// TIA Portal project "FactoryIO_Template_S7-1200_V15_V16" (V16)
// Vorlageprojekt für das Buch mit Zielsystem S7-1200

(* hardware
DEVICE "S7-1200-Station_1"  S7-1200 Station
   slot 0: "Baugruppenträger_0"  Rack  V1.0
   slot 1: "PLC_1"  CPU 1214C DC/DC/Rly  6ES7 214-1HG40-0XB0  V4.4
   slot 2: "DQ 16x24VDC_1"  SM 1222 DQ16 x 24VDC  6ES7 222-1BH32-0XB0  V2.0
*)

// ===== PLC "PLC_1"  CPU 1214C DC/DC/Rly =====

VAR_GLOBAL   // PLC tag table "Standard-Variablentabelle"
   "system" AT %M0.0 : Bool;
   "small_box_sensor_memory" AT %M0.1 : Bool;
   "large_box_sensor_memory" AT %M0.2 : Bool;
   "Transfer Right" AT %Q1.0 : Bool;
   "Tag_1" AT %M0.3 : Bool;
   "Tag_2" AT %M0.4 : Bool;
END_VAR

VAR_GLOBAL   // PLC tag table "Tag table from XML_1"
   "Start Button 1" AT %I0.0 : Bool;
   "Stop Button 1" AT %I0.1 : Bool;
   "Reset Button 1" AT %I0.2 : Bool;
   "Emergency Stop 1" AT %I0.3 : Bool;
   "input sensor" AT %I0.4 : Bool;
   "Roller Limit Sensor" AT %I0.5 : Bool;
   "Left Conveyor Sensor" AT %I0.6 : Bool;
   "Right Conveyor Sensor" AT %I0.7 : Bool;
   "Left Conveyor End Sensor" AT %I1.0 : Bool;
   "Right Conveyor End Sensor" AT %I1.1 : Bool;
   "Small Box Sensor" AT %I1.2 : Bool;
   "Large Box Sensor" AT %I1.3 : Bool;
   "Start Button Light" AT %Q0.0 : Bool;
   "Stop Button Light" AT %Q0.1 : Bool;
   "Reset Button Light" AT %Q0.2 : Bool;
   "Roller Conveyor (4m) 1" AT %Q0.3 : Bool;
   "Roller Conveyor (4m) 2" AT %Q0.4 : Bool;
   "Roller Conveyor (4m) 3" AT %Q0.5 : Bool;
   "roll forward" AT %Q0.6 : Bool;
   "Transfer Left" AT %Q0.7 : Bool;
   "Small Box Counter" AT %QD8 : DInt;
   "Large Box Counter" AT %QD12 : DInt;
END_VAR

// folder: System blocks/Program resources

DATA_BLOCK "IEC_Counter_0_DB"   // DB1
{ S7_Optimized_Access := 'TRUE' }
AUTHOR : Simatic
FAMILY : IEC
NAME : CNTR
VERSION : 1.0
// stored: InstanceOfName IEC_COUNTER
"IEC_COUNTER"
BEGIN
END_DATA_BLOCK

DATA_BLOCK "timer 2"   // DB2
{ S7_Optimized_Access := 'TRUE' }
AUTHOR : Simatic
FAMILY : IEC
NAME : IEC_TMR
VERSION : 1.0
// stored: InstanceOfName IEC_TIMER
"IEC_TIMER"
BEGIN
END_DATA_BLOCK

DATA_BLOCK "timer 1"   // DB3
{ S7_Optimized_Access := 'TRUE' }
AUTHOR : Simatic
FAMILY : IEC
NAME : IEC_TMR
VERSION : 1.0
// stored: InstanceOfName IEC_TIMER
"IEC_TIMER"
BEGIN
END_DATA_BLOCK

DATA_BLOCK "Counter 2"   // DB4
{ S7_Optimized_Access := 'TRUE' }
AUTHOR : Simatic
FAMILY : IEC
NAME : CNTR
VERSION : 1.0
// stored: InstanceOfName IEC_COUNTER
"IEC_COUNTER"
BEGIN
END_DATA_BLOCK

// folder: (top level)

FUNCTION "MHJ-PLC-Lab-Function-S71200" : Void   // FC9000, SCL
{ S7_Optimized_Access := 'TRUE' }
VERSION : 0.1
   VAR_TEMP
      rdTimeReturn : Int;
      outputTime : DTL;
      SyncVal : Byte;
      forVal : Int;
      forVal_2 : Int;
      Value : Byte;
   END_VAR
   VAR CONSTANT
      CompVal : Byte := 16#34;
      Value_01 : Byte := 16#11;
      Value_01_DW : DWord := 16#A165_D992;
      Value_02_DW : DWord := 16#58BE_4401;
   END_VAR
BEGIN

   #Value:=PEEK(area := 16#82,
        dbNumber := 0,
        byteOffset := 511);
   #Value := #Value + 1;

   POKE(area := 16#82,
        dbNumber := 0,
        byteOffset := 511,
        value := #Value);

   POKE(area:=16#81,
        dbNumber:=0,
        byteOffset:=1016,
        value:=#Value_01_DW);
   POKE(area := 16#81,
        dbNumber := 0,
        byteOffset := 1020,
        value := #Value_02_DW);

   POKE(area := 16#81,
        dbNumber := 0,
        byteOffset := 511,
        value := B#16#00);

   FOR #forVal := 0 TO 120 DO
       FOR #forVal_2:=0 TO 10 DO
           #rdTimeReturn:=RD_SYS_T(#outputTime);
           #rdTimeReturn := WR_SYS_T(#outputTime);
           #rdTimeReturn := RD_SYS_T(#outputTime);
           #rdTimeReturn := WR_SYS_T(#outputTime);
       END_FOR;
       #SyncVal:= PEEK(area := 16#81,
                      dbNumber := 0,
                      byteOffset := 511);
       IF #SyncVal = #CompVal THEN
          GOTO M_1;
       END_IF;
   END_FOR;
   RETURN;

   M_1:
   POKE(area := 16#81,
        dbNumber := 0,
        byteOffset := 511,
        value := B#16#0);
END_FUNCTION

ORGANIZATION_BLOCK "Main"   // OB1, LAD, ProgramCycle
TITLE = "Main Program Sweep (Cycle)"
{ S7_Optimized_Access := 'TRUE' }
VERSION : 0.1
   VAR_INPUT
      Initial_Call : Bool;   // Initial call of this OB
      Remanence : Bool;   // =True, if remanent data are available
   END_VAR
   VAR_TEMP   // added for the SCL form of the ladder/FBD networks
      _w1 : Bool;
   END_VAR
BEGIN

REGION Network 1: Konnektierungsbaustein für PLC-Lab
   // Im Netzwerk 1 wird der Konnektierungsbaustein für PLC-Lab aufgerufen.
   // Dieser Aufruf darf nicht entfernt werden!
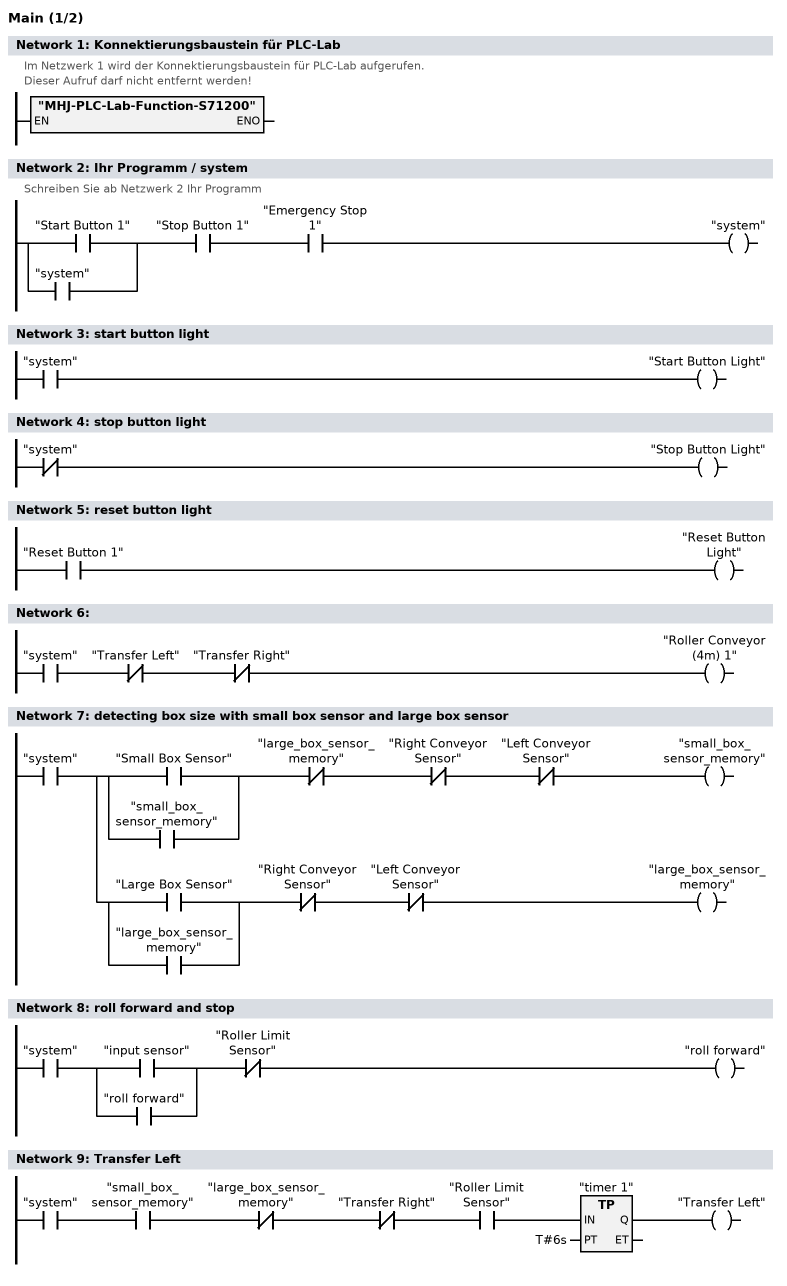
   RUNG wire#powerrail
      "MHJ-PLC-Lab-Function-S71200"()
   END_RUNG
   // the same network as SCL:
   "MHJ-PLC-Lab-Function-S71200"();
END_REGION

REGION Network 2: Ihr Programm / system
   // Schreiben Sie ab Netzwerk 2 Ihr Programm
   RUNG wire#powerrail
      Contact( "Start Button 1" )
      wire#w1
      Contact( "Stop Button 1" )
      Contact( "Emergency Stop 1" )
      Coil( "system" )
   END_RUNG
   RUNG wire#powerrail
      Contact( "system" )
   END_RUNG wire#w1
   // the same network as SCL:
   "system" := ("Start Button 1" OR "system") AND "Stop Button 1" AND "Emergency Stop 1";
END_REGION

REGION Network 3: start button light
   RUNG wire#powerrail
      Contact( "system" )
      Coil( "Start Button Light" )
   END_RUNG
   // the same network as SCL:
   "Start Button Light" := "system";
END_REGION

REGION Network 4: stop button light
   RUNG wire#powerrail
      I_Contact( "system" )
      Coil( "Stop Button Light" )
   END_RUNG
   // the same network as SCL:
   "Stop Button Light" := NOT "system";
END_REGION

REGION Network 5: reset button light
   RUNG wire#powerrail
      Contact( "Reset Button 1" )
      Coil( "Reset Button Light" )
   END_RUNG
   // the same network as SCL:
   "Reset Button Light" := "Reset Button 1";
END_REGION

REGION Network 6
   RUNG wire#powerrail
      Contact( "system" )
      I_Contact( "Transfer Left" )
      I_Contact( "Transfer Right" )
      Coil( "Roller Conveyor (4m) 1" )
   END_RUNG
   // the same network as SCL:
   "Roller Conveyor (4m) 1" := "system" AND NOT "Transfer Left" AND NOT "Transfer Right";
END_REGION

REGION Network 7: detecting box size with small box sensor and large box sensor
   RUNG wire#powerrail
      Contact( "system" )
      wire#w1
      Contact( "Small Box Sensor" )
      wire#w2
      I_Contact( "large_box_sensor_memory" )
      I_Contact( "Right Conveyor Sensor" )
      I_Contact( "Left Conveyor Sensor" )
      Coil( "small_box_sensor_memory" )
   END_RUNG
   RUNG wire#w1
      Contact( "small_box_sensor_memory" )
   END_RUNG wire#w2
   RUNG wire#w1
      Contact( "Large Box Sensor" )
      wire#w3
      I_Contact( "Right Conveyor Sensor" )
      I_Contact( "Left Conveyor Sensor" )
      Coil( "large_box_sensor_memory" )
   END_RUNG
   RUNG wire#w1
      Contact( "large_box_sensor_memory" )
   END_RUNG wire#w3
   // the same network as SCL:
   "small_box_sensor_memory" := "system" AND ("Small Box Sensor" OR "small_box_sensor_memory") AND NOT "large_box_sensor_memory" AND NOT "Right Conveyor Sensor" AND NOT "Left Conveyor Sensor";
   "large_box_sensor_memory" := "system" AND ("Large Box Sensor" OR "large_box_sensor_memory") AND NOT "Right Conveyor Sensor" AND NOT "Left Conveyor Sensor";
END_REGION

REGION Network 8: roll forward and stop
   RUNG wire#powerrail
      Contact( "system" )
      wire#w1
      Contact( "input sensor" )
      wire#w2
      I_Contact( "Roller Limit Sensor" )
      Coil( "roll forward" )
   END_RUNG
   RUNG wire#w1
      Contact( "roll forward" )
   END_RUNG wire#w2
   // the same network as SCL:
   "roll forward" := "system" AND ("input sensor" OR "roll forward") AND NOT "Roller Limit Sensor";
END_REGION

REGION Network 9: Transfer Left
   "timer 1".TP(IN := "system" AND "small_box_sensor_memory" AND NOT "large_box_sensor_memory" AND NOT "Transfer Right" AND "Roller Limit Sensor",
                PT := T#6s);
   "Transfer Left" := "timer 1".Q;
END_REGION

REGION Network 10: Transfer Left
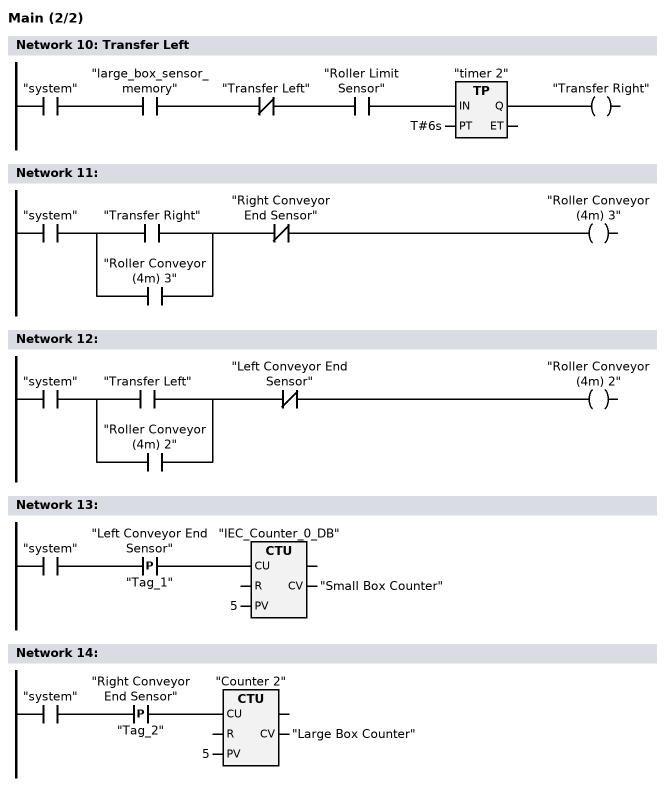
   "timer 2".TP(IN := "system" AND "large_box_sensor_memory" AND NOT "Transfer Left" AND "Roller Limit Sensor",
                PT := T#6s);
   "Transfer Right" := "timer 2".Q;
END_REGION

REGION Network 11
   RUNG wire#powerrail
      Contact( "system" )
      wire#w1
      Contact( "Transfer Right" )
      wire#w2
      I_Contact( "Right Conveyor End Sensor" )
      Coil( "Roller Conveyor (4m) 3" )
   END_RUNG
   RUNG wire#w1
      Contact( "Roller Conveyor (4m) 3" )
   END_RUNG wire#w2
   // the same network as SCL:
   "Roller Conveyor (4m) 3" := "system" AND ("Transfer Right" OR "Roller Conveyor (4m) 3") AND NOT "Right Conveyor End Sensor";
END_REGION

REGION Network 12
   RUNG wire#powerrail
      Contact( "system" )
      wire#w1
      Contact( "Transfer Left" )
      wire#w2
      I_Contact( "Left Conveyor End Sensor" )
      Coil( "Roller Conveyor (4m) 2" )
   END_RUNG
   RUNG wire#w1
      Contact( "Roller Conveyor (4m) 2" )
   END_RUNG wire#w2
   // the same network as SCL:
   "Roller Conveyor (4m) 2" := "system" AND ("Transfer Left" OR "Roller Conveyor (4m) 2") AND NOT "Left Conveyor End Sensor";
END_REGION

REGION Network 13
   #_w1 := "system" AND "Left Conveyor End Sensor" AND NOT "Tag_1";   // rising edge of "Left Conveyor End Sensor"
   "Tag_1" := "Left Conveyor End Sensor";
   "IEC_Counter_0_DB".CTU(CU := #_w1, PV := 5, CV => "Small Box Counter");
END_REGION

REGION Network 14
   #_w1 := "system" AND "Right Conveyor End Sensor" AND NOT "Tag_2";   // rising edge of "Right Conveyor End Sensor"
   "Tag_2" := "Right Conveyor End Sensor";
   "Counter 2".CTU(CU := #_w1, PV := 5, CV => "Large Box Counter");
END_REGION
END_ORGANIZATION_BLOCK